FUNCTION_BLOCK FB_READ_HW
VAR_INPUT
END_VAR
VAR_OUTPUT
END_VAR
VAR
END_VAR

(*READ HARDWARE FUCNTION BLOCK

	Reads all variables from devices on the EtherCAT network and
	assigns them to their relevant program variables.  This will
	happen every PLC scan*)

(*Left Drive Motor*)
//HARV.DriveSys.DriveLeftIN.ActualVelocity := MOTORS.DriveLeft.ActualVelocity;
HARV.DriveSys.DriveLeftIN.StatusWord 			:= MOTORS.DriveLeft.StatusWord;
HARV.DriveSys.DriveLeftIN.ActualVelocity 		:= MOTORS.DriveLeft.ActualVelocity;
HARV.DriveSys.DriveLeftIN.BatteryVoltage		:= MOTORS.DriveLeft.BatteryVoltage;
HARV.DriveSys.DriveLeftIN.BatteryCurrent		:= MOTORS.DriveLeft.BatteryCurrent;
HARV.DriveSys.DriveLeftIN.HeatSinkTemp			:= MOTORS.DriveLeft.HeatsinkTemp;
HARV.DriveSys.DriveLeftIN.CapacitorVoltage		:= MOTORS.DriveLeft.CapacitorVoltage;

(*Right Drive Motor*)
HARV.DriveSys.DriveRightIN.StatusWord			:= MOTORS.DriveRight.StatusWord;
HARV.DriveSys.DriveRightIN.ActualVelocity 		:= MOTORS.DriveRight.ActualVelocity;
HARV.DriveSys.DriveRightIN.BatteryVoltage		:= MOTORS.DriveRight.BatteryVoltage;
HARV.DriveSys.DriveRightIN.BatteryCurrent		:= MOTORS.DriveRight.BatteryCurrent;
HARV.DriveSys.DriveRightIN.HeatSinkTemp			:= MOTORS.DriveRight.HeatsinkTemp;
HARV.DriveSys.DriveRightIN.CapacitorVoltage		:= MOTORS.DriveRight.CapacitorVoltage;

(*Left Steering Motor*)
HARV.DriveSys.SteerLeftIN.StatusWord 			:= MOTORS.SteerLeft.StatusWord;
HARV.DriveSys.SteerLeftIN.ActualPosition 		:= MOTORS.SteerLeft.ActualPosition;
HARV.DriveSys.SteerLeftIN.ActualVelocity 		:= MOTORS.SteerLeft.ActualVelocity;
HARV.DriveSys.SteerLeftIN.OperationModeDisplay 	:= MOTORS.SteerLeft.OperationModeDisplay;

(*Right Steering Motor*)
HARV.DriveSys.SteerRightIN.StatusWord 			:= MOTORS.SteerRight.StatusWord;
HARV.DriveSys.SteerRightIN.ActualPosition 		:= MOTORS.SteerRight.ActualPosition;
HARV.DriveSys.SteerRightIN.ActualVelocity 		:= MOTORS.SteerRight.ActualVelocity;
HARV.DriveSys.SteerRightIN.OperationModeDisplay := MOTORS.SteerRight.OperationModeDisplay;

(*Left Conveyance Motor*)

(*Right Conveyance Motor*)

(*Tilt Control Inputs*)

(*Digital Inputs EL1018*)
//HARV.DriveSys.JohnButtonInput := IO.DI_SLICE_0[0];
UI.PickButton := IO.DI_SLICE_0[0];
HARV.TiltControl.PressureSwitch := IO.DI_SLICE_0[1];
UI.EStop := IO.DI_SLICE_0[2];

(*Analog Inputs EL3064*)
HARV.DriveSys.JoyStick_X 		:= IO.AI_SLICE_0[0];
HARV.DriveSys.JoyStick_Y 		:= IO.AI_SLICE_0[1];
//HARV.DriveSys.JoyStick_Button 	:= IO.AI_SLICE_0[2];
HARV.TiltControl.IMU_Roll		:= IO.AI_SLICE_0[2];
HARV.TiltControl.IMU_Pitch		:= IO.AI_SLICE_0[3];

(**)

END_FUNCTION_BLOCK

(* stored: Version 1.1.0.1, ProductVersion 3.1.4024.12
   POU FB_READ_HW: Id {ac7844ff-7952-49bf-b678-2d246b8cfef7}, SpecialFunc None *)
